(* IEC 61131-3 sources: Industry-PLC-LLM/data/PLCBEAD_repo/PLCBEAD_PLCEmbed-main/PLC-BEAD/Source/GEB/_WORD_TO_REAL, 1 file *)

(* ---- _WORD_TO_REAL.ST ---- *)
FUNCTION _WORD_TO_REAL:REAL
	VAR_INPUT
		IN :	WORD;
	END_VAR
	_WORD_TO_REAL := UINT_TO_REAL(WORD_TO_UINT(IN));
END_FUNCTION

PROGRAM program0
  VAR
    LocalVar0 : WORD;
    LocalOUT  : REAL;
  END_VAR

  LocalOUT := _WORD_TO_REAL(LocalVar0);
END_PROGRAM
